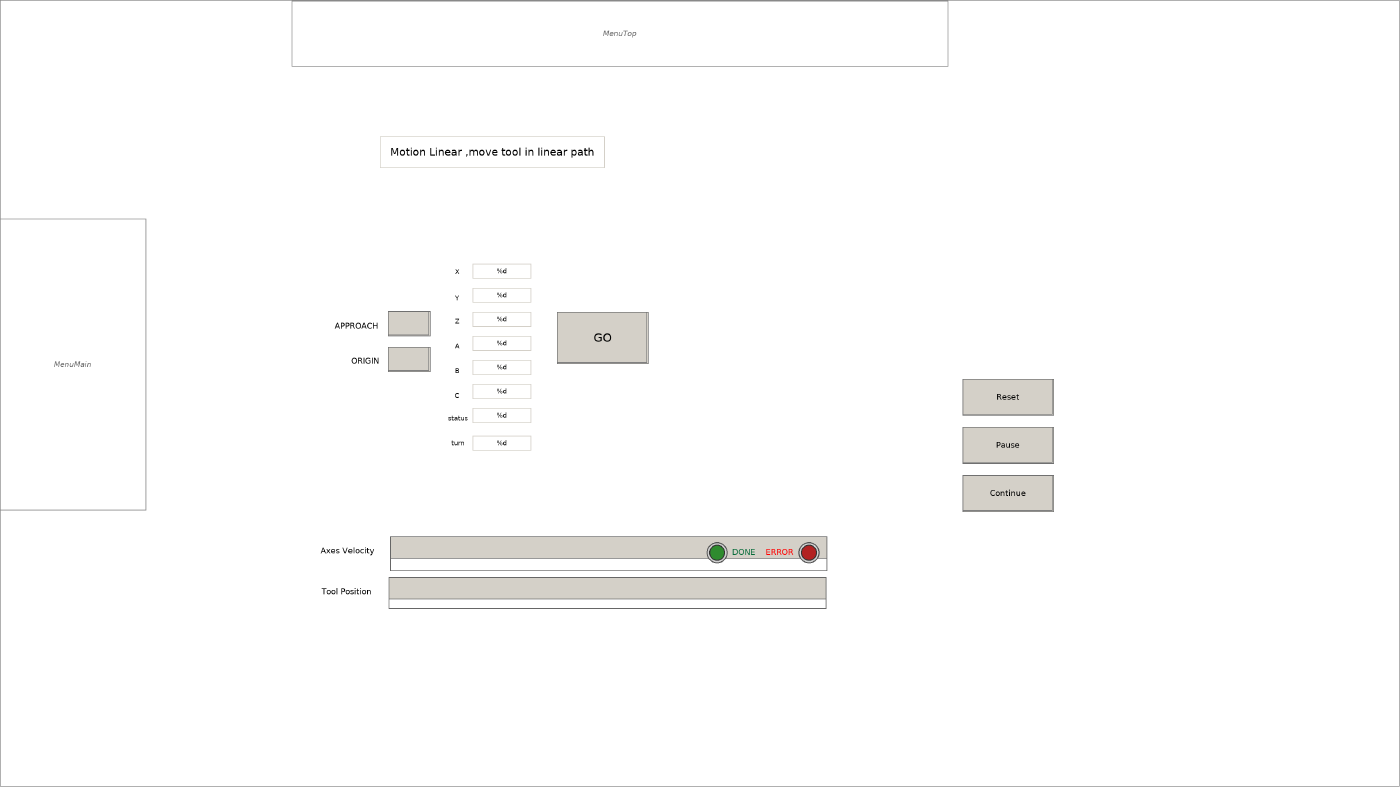
VISUALIZATION Motion_Linear  // 1920x1080
    Frame (400,1 900x90)
        shows MenuTop()
    Frame (0,300 200x400)
        shows MenuMain()
    Textfield (521,187 308x43), "Motion Linear ,move tool in linear path"
    Button (764,428 125x71), "GO"
        tap MAIN.Move_Linear.Execute
    Textfield (648,362 80x20), "%d", text variable: main.LinearTargetPOS.X
    Textfield (648,395 80x20), "%d", text variable: main.LinearTargetPOS.Y
    Textfield (648,428 80x20), "%d", text variable: main.LinearTargetPOS.Z
    Textfield (648,461 80x20), "%d", text variable: main.LinearTargetPOS.A
    Textfield (648,494 80x20), "%d", text variable: main.LinearTargetPOS.B
    Textfield (648,527 80x20), "%d", text variable: main.LinearTargetPOS.C
    Label (610,361 34x24), "X"
    Label (610,397 34x24), "Y"
    Label (610,429 34x24), "Z"
    Label (610,463 34x24), "A"
    Label (610,497 34x24), "B"
    Label (610,531 34x24), "C"
    Label (454,433 70x29), "APPROACH"
    Label (478,481 46x29), "ORIGIN"
    Button (532,427 58x34)
        OnMouseClick: execute {
            //APPROACH COORDINATES:
            main.LinearTargetPOS.X:=974.21;
            main.LinearTargetPOS.y:=-18.91;
            main.LinearTargetPOS.z:=1704.54;
            main.LinearTargetPOS.a:=-97.73;
            main.LinearTargetPOS.b:=88.22;
            main.LinearTargetPOS.c:=-96.10;
            main.LinearTargetPOS.Status :=18;
            main.LinearTargetPOS.Turn:=2;
            //approach
        }
    Button (532,476 58x34)
        OnMouseClick: execute {
            //origin
            main.LinearTargetPOS.X:=1486.29;
            main.LinearTargetPOS.y:=-26.88;
            main.LinearTargetPOS.z:=1422.08;
            main.LinearTargetPOS.a:=-98.31;
            main.LinearTargetPOS.b:=88.04;
            main.LinearTargetPOS.c:=-96.97;
            main.LinearTargetPOS.Status :=18;
            main.LinearTargetPOS.Turn:=2;
        }
    Label (621,326 112x24)
    Textfield (648,560 80x20), "%d", text variable: main.LinearTargetPOS.Status
    Textfield (648,598 80x20), "%d", text variable: main.LinearTargetPOS.Turn
    Label (611,562 34x24), "status"
    Label (611,596 34x24), "turn"
    Button (1320,586 125x50), "Pause"
        tap mxA_Motion.fbAutoDemo.fbKRC_Interrupt.Execute
    Button (1320,652 125x50), "Continue"
        tap mxA_Motion.fbAutoDemo.fbKRC_Continue.Enable
    Button (1320,520 125x50), "Reset"
        tap MAIN.Write_Program_Abort.ExecuteCmd
    Table (533,792 600x43), data array: mxA_Motion.fbKRC_ReadActualPosition.Position
        p3854506369: mxA_Motion.fbKRC_ReadActualPosition.Position.X
        p1892666644: mxA_Motion.fbKRC_ReadActualPosition.Position.Y
        p338671338: mxA_Motion.fbKRC_ReadActualPosition.Position.Z
        p2170511999: mxA_Motion.fbKRC_ReadActualPosition.Position.A
        p3723444502: mxA_Motion.fbKRC_ReadActualPosition.Position.B
        p1218418051: mxA_Motion.fbKRC_ReadActualPosition.Position.C
        p746581629: mxA_Motion.fbKRC_ReadActualPosition.Position.Status
        p3104783080: mxA_Motion.fbKRC_ReadActualPosition.Position.Turn
        p2501879983: mxA_Motion.fbKRC_ReadActualPosition.Position.E1
        p7306298: mxA_Motion.fbKRC_ReadActualPosition.Position.E2
        p1933151965: mxA_Motion.fbKRC_ReadActualPosition.Position.E3
        p3863566920: mxA_Motion.fbKRC_ReadActualPosition.Position.E4
        p2192122294: mxA_Motion.fbKRC_ReadActualPosition.Position.E5
        p400160035: mxA_Motion.fbKRC_ReadActualPosition.Position.E6
        p1757482276: status
        p4088588272: turn
    Table (535,736 599x47), data array: Read_Axes_Velocity.ReadAxesVelocity
        p3854506369: Read_Axes_Velocity.ReadAxesVelocity.AxisGroupIdx
        p1892666644: Read_Axes_Velocity.ReadAxesVelocity.ExecuteCmd
        p338671338: Read_Axes_Velocity.ReadAxesVelocity.Done
        p2170511999: Read_Axes_Velocity.ReadAxesVelocity.Error
        p3723444502: Read_Axes_Velocity.ReadAxesVelocity.ErrorID
        p1218418051: Read_Axes_Velocity.ReadAxesVelocity.A1
        p746581629: Read_Axes_Velocity.ReadAxesVelocity.A2
        p3104783080: Read_Axes_Velocity.ReadAxesVelocity.A3
        p2501879983: Read_Axes_Velocity.ReadAxesVelocity.A4
        p7306298: Read_Axes_Velocity.ReadAxesVelocity.A5
        p1933151965: Read_Axes_Velocity.ReadAxesVelocity.A6
        p3863566920: Read_Axes_Velocity.ReadAxesVelocity.E1
        p2192122294: Read_Axes_Velocity.ReadAxesVelocity.E2
        p400160035: Read_Axes_Velocity.ReadAxesVelocity.E3
        p1265227338: Read_Axes_Velocity.ReadAxesVelocity.E4
        p3726181087: Read_Axes_Velocity.ReadAxesVelocity.E5
        p3136911649: Read_Axes_Velocity.ReadAxesVelocity.E6
        p797552052: Read_Axes_Velocity.ReadAxesVelocity.mxA_ExecuteCommand
    Rectangle (430,741 93x30), "Axes Velocity"
    Lamp1 (967,742 33x33), variable: Read_Axes_Velocity.ReadAxesVelocity.Done, style: Lamp-Lamp1-Green
    Lamp1 (1093,742 33x33), variable: Read_Axes_Velocity.ReadAxesVelocity.Error, style: Lamp-Lamp1-Red
    Rectangle (997,747 46x22), "DONE"
    Rectangle (1046,747 46x22), "ERROR"
    Rectangle (429,797 93x30), "Tool Position"
END_VISUALIZATION

(* stored: Version 1.1.0.1, ProductVersion 3.1.4024.10
   Visu Motion_Linear: Id {3cfb20d2-caa8-4d81-bcca-d8a3f923c164} *)
